(* Logix 5000 project; controller ProjectTemplate vendor 1 type 14 code 213 rev 35.11; software revision 35.01 *)

TASK SafetyTask (periodic, rate 20 ms, priority 10, watchdog 20 ms, safety)

MODULES
   Local : vendor 1 type 14 code 213 (ICP 0, rev 35.11)
END_MODULES
